/// Link to Lisec [Lisec](https://www.lisec.com)
///![Lisec](../images/logo.png)
/// This a empty **POU**
PROGRAM POU
VAR
	i : INT;
END_VAR

METHOD ABSTRACT M_Test1 : BOOL
VAR_INPUT
	sTest1 : T_MaxString;
	nTest2 : LREAL;
END_VAR
END_METHOD

PROPERTY PROTECTED ABSTRACT P_BAR : BOOL
GET
END_GET
SET
END_SET
END_PROPERTY

END_PROGRAM

(* stored: Version 1.1.0.1
   POU POU: Id {69af5d91-944a-455f-89fd-cdceba92cb5b}, SpecialFunc None
   Method M_Test1: Id {d272ab2c-3a36-4b3d-a06c-8c9ae873ad4a}
   Property P_BAR: Id {8f3d2245-d837-4ab1-b994-b57d7e7feedb}
   Get Get: Id {1da35c9b-b2b9-4e21-862c-4a736b41de91}
   Set Set: Id {8a08dd1a-0de4-4cc7-b524-c71296317bff} *)
